{attribute 'GeneratedUsingTerminal: EP6228-0042-0016'}
{attribute addProperty BoxType "EP6228-0042-0016"}
{attribute addProperty Id "Module_1_DeviceState_Inputs_DeviceModule_1_DeviceState_Inputs_Device_5322301C2Module_2_DeviceState_InputsModule_2_DeviceState_Inputs_B92A0D6A8Module_11_Digital_InputsModule_11_Digital_Inputs_33FD83728WcStateAT %I*WcState_9091E0EB2InfoDataAT %I*InfoData_90184F0C16"}
{attribute addProperty CRC "1230723316"}
{attribute addProperty Size "36"}
TYPE EP6228_495B58F4 EXTENDS EtcSlaveTerminalBase_947E5A46 :
STRUCT
	{attribute addProperty Name "Module_1_DeviceState_Inputs_Device"}
	Module_1_DeviceState_Inputs_Device : Module_1_DeviceState_Inputs_Device_5322301C;
	{attribute addProperty Name "Module_2_DeviceState_Inputs"}
	Module_2_DeviceState_Inputs : Module_2_DeviceState_Inputs_B92A0D6A;
	{attribute addProperty Name "Module_11_Digital_Inputs"}
	Module_11_Digital_Inputs : Module_11_Digital_Inputs_33FD8372;
	{attribute addProperty Name "WcState"}
	WcState : WcState_9091E0EB;
	{attribute addProperty Name "InfoData"}
	InfoData : InfoData_90184F0C;
END_STRUCT
END_TYPE

(* stored: Version 1.2.0.0, ProductVersion 3.1.4024.9
   DUT EP6228_495B58F4: Id {0c532096-0954-4e7e-8977-31cd8de73a24} *)
